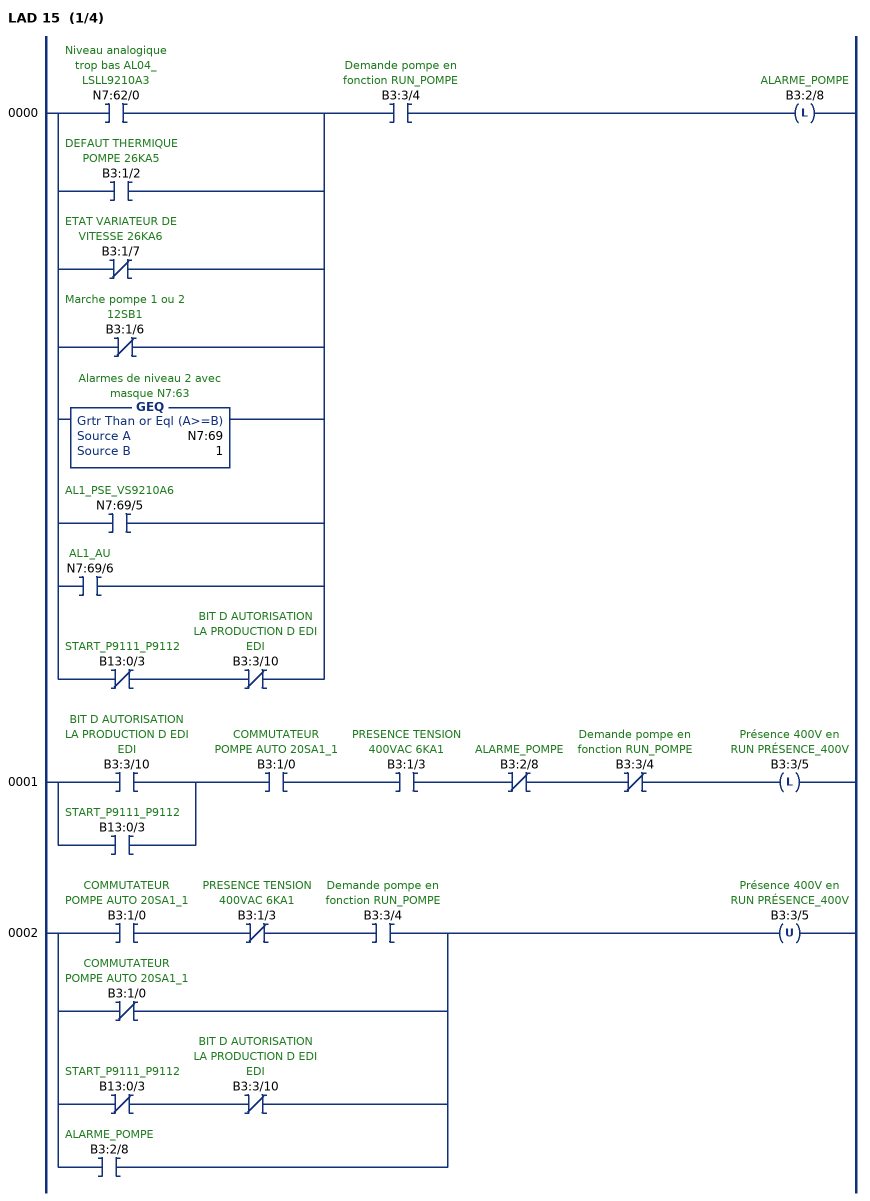
% Rung: 0 %
SOR BST XIC N7:62/0 NXB XIC B3:1/2 NXB XIO B3:1/7 NXB XIO B3:1/6 NXB GEQ N7:69 1 NXB XIC N7:69/5 NXB XIC N7:69/6 NXB XIO B13:0/3 XIO B3:3/10 BND XIC B3:3/4 OTL B3:2/8 EOR
%   N7:62/0  AL04_LSLL9210A3  "Niveau analogique trop bas" %
%   B3:1/2  26KA5  "DEFAUT THERMIQUE POMPE" %
%   B3:1/7  26KA6  "ETAT VARIATEUR DE VITESSE" %
%   B3:1/6  12SB1  "Marche pompe 1 ou 2" %
%   N7:69  "Alarmes de niveau 2 avec masque N7:63" %
%   N7:69/5  AL1_PSE_VS9210A6 %
%   N7:69/6  AL1_AU %
%   B13:0/3  START_P9111_P9112 %
%   B3:3/10  EDI  "BIT D AUTORISATION LA PRODUCTION D EDI" %
%   B3:3/4  RUN_POMPE  "Demande pompe en fonction" %
%   B3:2/8  ALARME_POMPE %
% Rung: 1 %
SOR BST XIC B3:3/10 NXB XIC B13:0/3 BND XIC B3:1/0 XIC B3:1/3 XIO B3:2/8 XIO B3:3/4 OTL B3:3/5 EOR
%   B3:3/10  EDI  "BIT D AUTORISATION LA PRODUCTION D EDI" %
%   B13:0/3  START_P9111_P9112 %
%   B3:1/0  20SA1_1  "COMMUTATEUR POMPE AUTO" %
%   B3:1/3  6KA1  "PRESENCE TENSION 400VAC" %
%   B3:2/8  ALARME_POMPE %
%   B3:3/4  RUN_POMPE  "Demande pompe en fonction" %
%   B3:3/5  PRÉSENCE_400V  "Présence 400V en RUN" %
% Rung: 2 %
SOR BST XIC B3:1/0 XIO B3:1/3 XIC B3:3/4 NXB XIO B3:1/0 NXB XIO B13:0/3 XIO B3:3/10 NXB XIC B3:2/8 BND OTU B3:3/5 EOR
%   B3:1/0  20SA1_1  "COMMUTATEUR POMPE AUTO" %
%   B3:1/3  6KA1  "PRESENCE TENSION 400VAC" %
%   B3:3/4  RUN_POMPE  "Demande pompe en fonction" %
%   B13:0/3  START_P9111_P9112 %
%   B3:3/10  EDI  "BIT D AUTORISATION LA PRODUCTION D EDI" %
%   B3:2/8  ALARME_POMPE %
%   B3:3/5  PRÉSENCE_400V  "Présence 400V en RUN" %

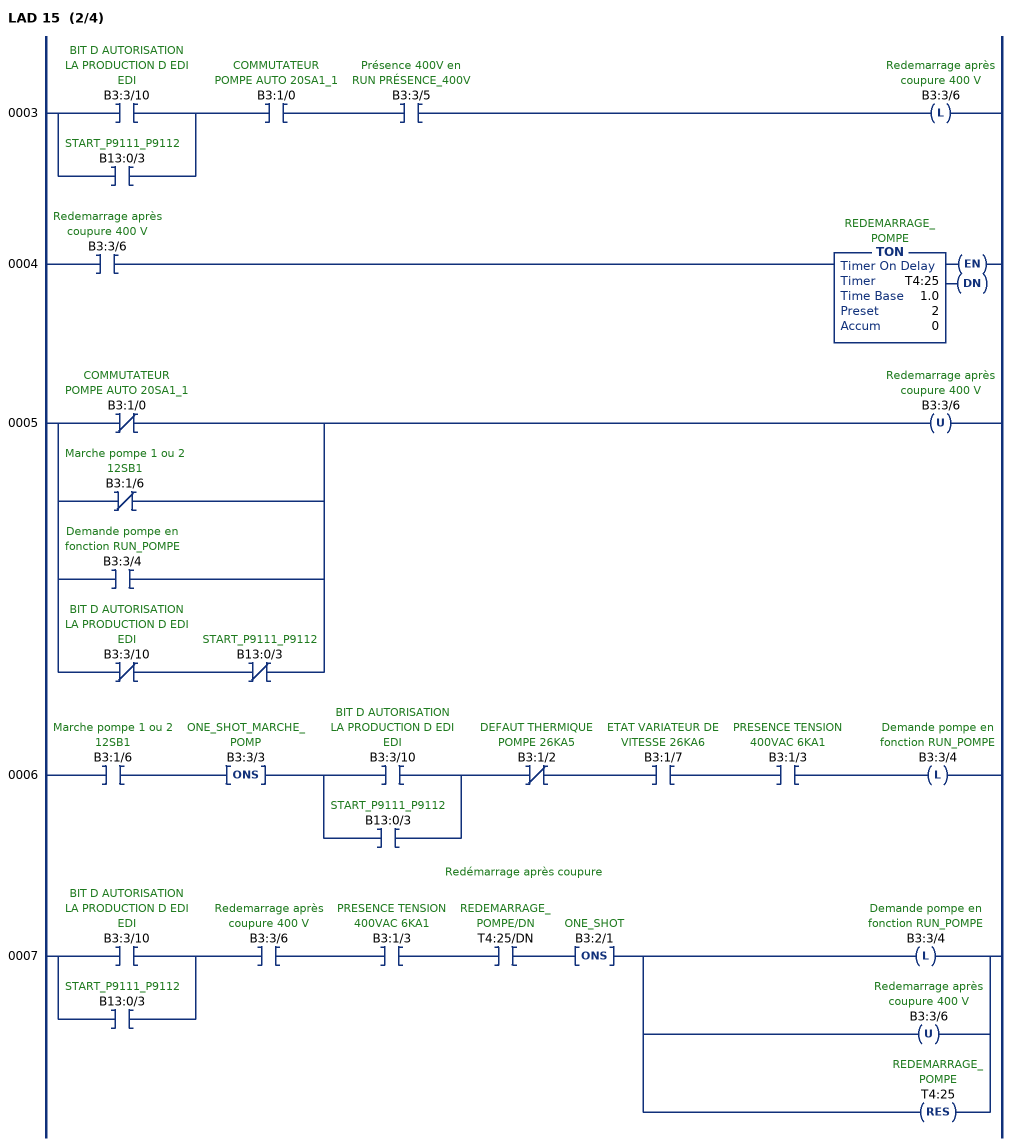
% Rung: 3 %
SOR BST XIC B3:3/10 NXB XIC B13:0/3 BND XIC B3:1/0 XIC B3:3/5 OTL B3:3/6 EOR
%   B3:3/10  EDI  "BIT D AUTORISATION LA PRODUCTION D EDI" %
%   B13:0/3  START_P9111_P9112 %
%   B3:1/0  20SA1_1  "COMMUTATEUR POMPE AUTO" %
%   B3:3/5  PRÉSENCE_400V  "Présence 400V en RUN" %
%   B3:3/6  "Redemarrage après coupure 400 V" %
% Rung: 4 %
SOR XIC B3:3/6 TON T4:25 1.0 2 0 EOR
%   B3:3/6  "Redemarrage après coupure 400 V" %
%   T4:25  REDEMARRAGE_POMPE %
% Rung: 5 %
SOR BST XIO B3:1/0 NXB XIO B3:1/6 NXB XIC B3:3/4 NXB XIO B3:3/10 XIO B13:0/3 BND OTU B3:3/6 EOR
%   B3:1/0  20SA1_1  "COMMUTATEUR POMPE AUTO" %
%   B3:1/6  12SB1  "Marche pompe 1 ou 2" %
%   B3:3/4  RUN_POMPE  "Demande pompe en fonction" %
%   B3:3/10  EDI  "BIT D AUTORISATION LA PRODUCTION D EDI" %
%   B13:0/3  START_P9111_P9112 %
%   B3:3/6  "Redemarrage après coupure 400 V" %
% Rung: 6 %
SOR XIC B3:1/6 OSR B3:3/3 BST XIC B3:3/10 NXB XIC B13:0/3 BND XIO B3:1/2 XIC B3:1/7 XIC B3:1/3 OTL B3:3/4 EOR
%   B3:1/6  12SB1  "Marche pompe 1 ou 2" %
%   B3:3/3  ONE_SHOT_MARCHE_POMP %
%   B3:3/10  EDI  "BIT D AUTORISATION LA PRODUCTION D EDI" %
%   B13:0/3  START_P9111_P9112 %
%   B3:1/2  26KA5  "DEFAUT THERMIQUE POMPE" %
%   B3:1/7  26KA6  "ETAT VARIATEUR DE VITESSE" %
%   B3:1/3  6KA1  "PRESENCE TENSION 400VAC" %
%   B3:3/4  RUN_POMPE  "Demande pompe en fonction" %
% Rung: 7 %
% Redémarrage après coupure %
SOR BST XIC B3:3/10 NXB XIC B13:0/3 BND XIC B3:3/6 XIC B3:1/3 XIC T4:25/DN OSR B3:2/1 BST OTL B3:3/4 NXB OTU B3:3/6 NXB RES T4:25 BND EOR
%   B3:3/10  EDI  "BIT D AUTORISATION LA PRODUCTION D EDI" %
%   B13:0/3  START_P9111_P9112 %
%   B3:3/6  "Redemarrage après coupure 400 V" %
%   B3:1/3  6KA1  "PRESENCE TENSION 400VAC" %
%   T4:25  REDEMARRAGE_POMPE %
%   B3:2/1  ONE_SHOT %
%   B3:3/4  RUN_POMPE  "Demande pompe en fonction" %

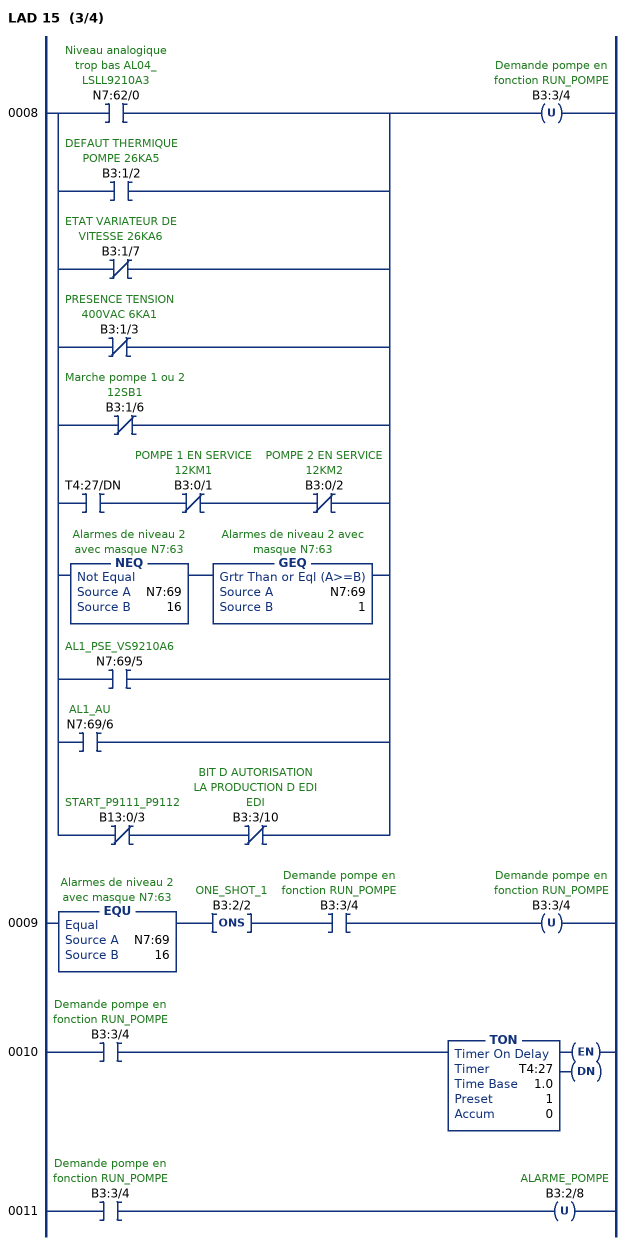
% Rung: 8 %
SOR BST XIC N7:62/0 NXB XIC B3:1/2 NXB XIO B3:1/7 NXB XIO B3:1/3 NXB XIO B3:1/6 NXB XIC T4:27/DN XIO B3:0/1 XIO B3:0/2 NXB NEQ N7:69 16 GEQ N7:69 1 NXB XIC N7:69/5 NXB XIC N7:69/6 NXB XIO B13:0/3 XIO B3:3/10 BND OTU B3:3/4 EOR
%   N7:62/0  AL04_LSLL9210A3  "Niveau analogique trop bas" %
%   B3:1/2  26KA5  "DEFAUT THERMIQUE POMPE" %
%   B3:1/7  26KA6  "ETAT VARIATEUR DE VITESSE" %
%   B3:1/3  6KA1  "PRESENCE TENSION 400VAC" %
%   B3:1/6  12SB1  "Marche pompe 1 ou 2" %
%   B3:0/1  12KM1  "POMPE 1 EN SERVICE" %
%   B3:0/2  12KM2  "POMPE 2 EN SERVICE" %
%   N7:69  "Alarmes de niveau 2 avec masque N7:63" %
%   N7:69/5  AL1_PSE_VS9210A6 %
%   N7:69/6  AL1_AU %
%   B13:0/3  START_P9111_P9112 %
%   B3:3/10  EDI  "BIT D AUTORISATION LA PRODUCTION D EDI" %
%   B3:3/4  RUN_POMPE  "Demande pompe en fonction" %
% Rung: 9 %
SOR EQU N7:69 16 OSR B3:2/2 XIC B3:3/4 OTU B3:3/4 EOR
%   N7:69  "Alarmes de niveau 2 avec masque N7:63" %
%   B3:2/2  ONE_SHOT_1 %
%   B3:3/4  RUN_POMPE  "Demande pompe en fonction" %
% Rung: 10 %
SOR XIC B3:3/4 TON T4:27 1.0 1 0 EOR
%   B3:3/4  RUN_POMPE  "Demande pompe en fonction" %
% Rung: 11 %
SOR XIC B3:3/4 OTU B3:2/8 EOR
%   B3:3/4  RUN_POMPE  "Demande pompe en fonction" %
%   B3:2/8  ALARME_POMPE %

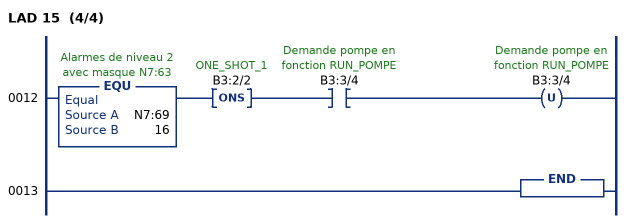
% Rung: 12 %
SOR EQU N7:69 16 OSR B3:2/2 XIC B3:3/4 OTU B3:3/4 EOR
%   N7:69  "Alarmes de niveau 2 avec masque N7:63" %
%   B3:2/2  ONE_SHOT_1 %
%   B3:3/4  RUN_POMPE  "Demande pompe en fonction" %
% Rung: 13 %
SOR END EOR

LADDER 16
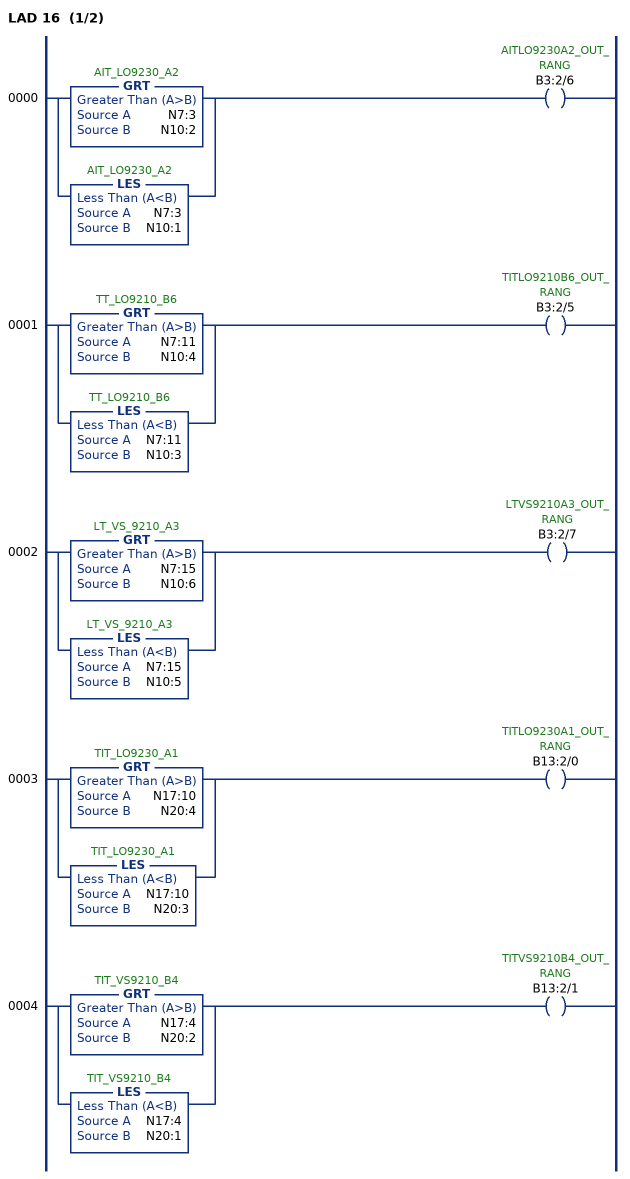
% Rung: 0 %
SOR BST GRT N7:3 N10:2 NXB LES N7:3 N10:1 BND OTE B3:2/6 EOR
%   N7:3  AIT_LO9230_A2 %
%   N10:2  OUT_RANG_MAX_AIT %
%   N10:1  OUT_RANG_MIN_AIT %
%   B3:2/6  AITLO9230A2_OUT_RANG %
% Rung: 1 %
SOR BST GRT N7:11 N10:4 NXB LES N7:11 N10:3 BND OTE B3:2/5 EOR
%   N7:11  TT_LO9210_B6 %
%   N10:4  OUT_RANG_MAX_TIT %
%   N10:3  OUT_RANG_MIN_TIT %
%   B3:2/5  TITLO9210B6_OUT_RANG %
% Rung: 2 %
SOR BST GRT N7:15 N10:6 NXB LES N7:15 N10:5 BND OTE B3:2/7 EOR
%   N7:15  LT_VS_9210_A3 %
%   N10:6  OUT_RANG_MAX_LT %
%   N10:5  OUT_RANG_MIN_LT %
%   B3:2/7  LTVS9210A3_OUT_RANG %
% Rung: 3 %
SOR BST GRT N17:10 N20:4 NXB LES N17:10 N20:3 BND OTE B13:2/0 EOR
%   N17:10  TIT_LO9230_A1 %
%   B13:2/0  TITLO9230A1_OUT_RANG %
% Rung: 4 %
SOR BST GRT N17:4 N20:2 NXB LES N17:4 N20:1 BND OTE B13:2/1 EOR
%   N17:4  TIT_VS9210_B4 %
%   B13:2/1  TITVS9210B4_OUT_RANG %

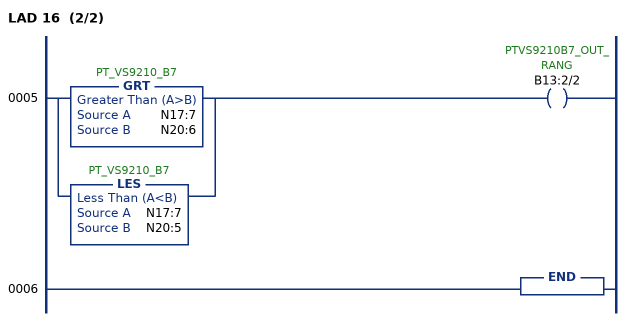
% Rung: 5 %
SOR BST GRT N17:7 N20:6 NXB LES N17:7 N20:5 BND OTE B13:2/2 EOR
%   N17:7  PT_VS9210_B7 %
%   B13:2/2  PTVS9210B7_OUT_RANG %
% Rung: 6 %
SOR END EOR

LADDER 17
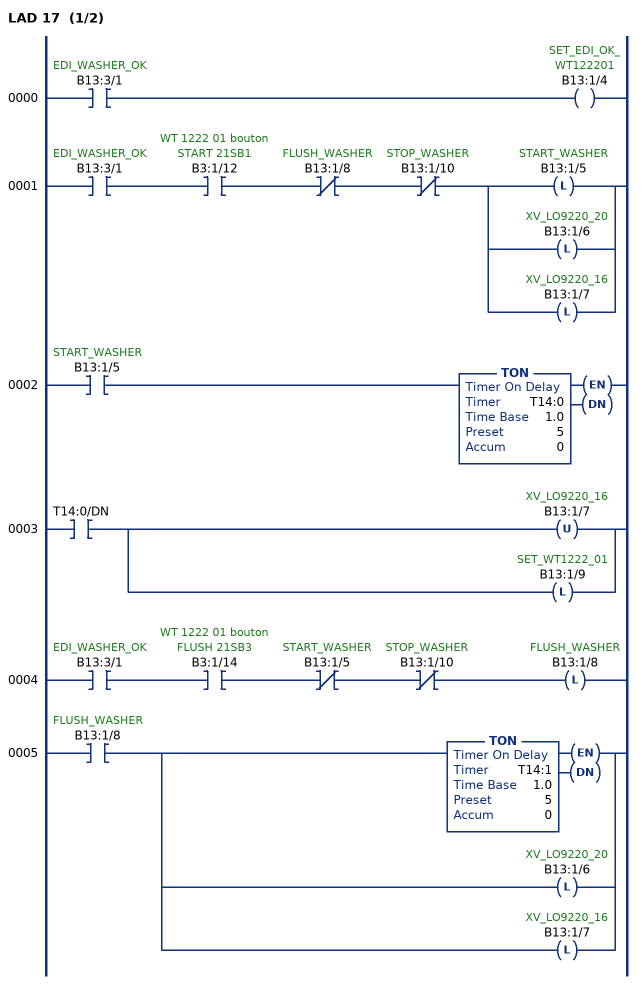
% Rung: 0 %
SOR XIC B13:3/1 OTE B13:1/4 EOR
%   B13:3/1  EDI_WASHER_OK %
%   B13:1/4  SET_EDI_OK_WT122201 %
% Rung: 1 %
SOR XIC B13:3/1 XIC B3:1/12 XIO B13:1/8 XIO B13:1/10 BST OTL B13:1/5 NXB OTL B13:1/6 NXB OTL B13:1/7 BND EOR
%   B13:3/1  EDI_WASHER_OK %
%   B3:1/12  21SB1  "WT 1222 01 bouton START" %
%   B13:1/8  FLUSH_WASHER %
%   B13:1/10  STOP_WASHER %
%   B13:1/5  START_WASHER %
%   B13:1/6  XV_LO9220_20 %
%   B13:1/7  XV_LO9220_16 %
% Rung: 2 %
SOR XIC B13:1/5 TON T14:0 1.0 5 0 EOR
%   B13:1/5  START_WASHER %
% Rung: 3 %
SOR XIC T14:0/DN BST OTU B13:1/7 NXB OTL B13:1/9 BND EOR
%   B13:1/7  XV_LO9220_16 %
%   B13:1/9  SET_WT1222_01 %
% Rung: 4 %
SOR XIC B13:3/1 XIC B3:1/14 XIO B13:1/5 XIO B13:1/10 OTL B13:1/8 EOR
%   B13:3/1  EDI_WASHER_OK %
%   B3:1/14  21SB3  "WT 1222 01 bouton FLUSH" %
%   B13:1/5  START_WASHER %
%   B13:1/10  STOP_WASHER %
%   B13:1/8  FLUSH_WASHER %
% Rung: 5 %
SOR XIC B13:1/8 BST TON T14:1 1.0 5 0 NXB OTL B13:1/6 NXB OTL B13:1/7 BND EOR
%   B13:1/8  FLUSH_WASHER %
%   B13:1/6  XV_LO9220_20 %
%   B13:1/7  XV_LO9220_16 %

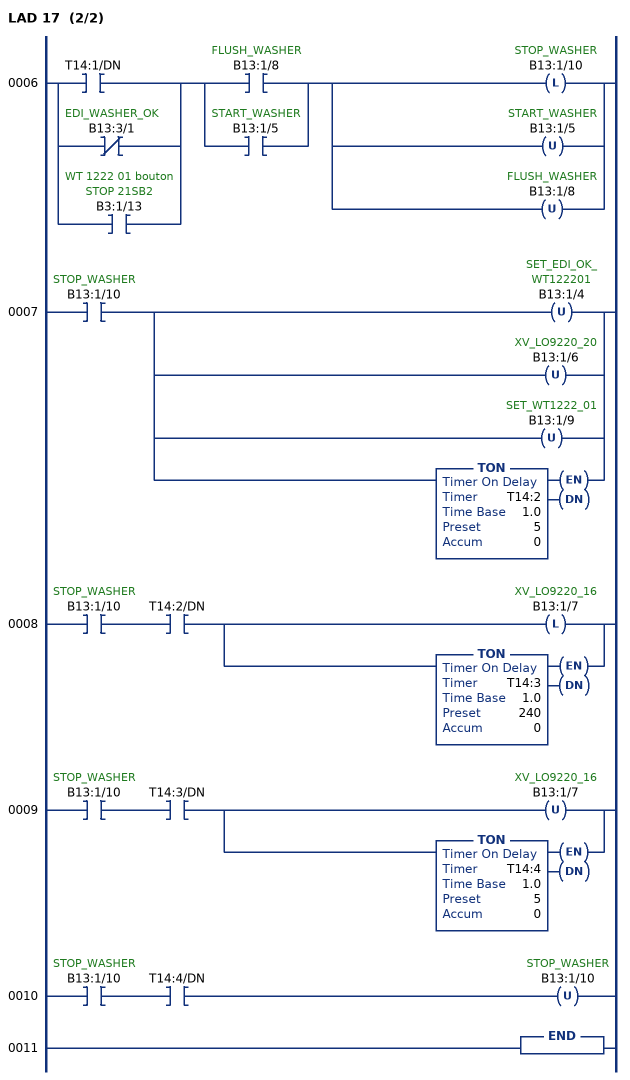
% Rung: 6 %
SOR BST XIC T14:1/DN NXB XIO B13:3/1 NXB XIC B3:1/13 BND BST XIC B13:1/8 NXB XIC B13:1/5 BND BST OTL B13:1/10 NXB OTU B13:1/5 NXB OTU B13:1/8 BND EOR
%   B13:3/1  EDI_WASHER_OK %
%   B3:1/13  21SB2  "WT 1222 01 bouton STOP" %
%   B13:1/8  FLUSH_WASHER %
%   B13:1/5  START_WASHER %
%   B13:1/10  STOP_WASHER %
% Rung: 7 %
SOR XIC B13:1/10 BST OTU B13:1/4 NXB OTU B13:1/6 NXB OTU B13:1/9 NXB TON T14:2 1.0 5 0 BND EOR
%   B13:1/10  STOP_WASHER %
%   B13:1/4  SET_EDI_OK_WT122201 %
%   B13:1/6  XV_LO9220_20 %
%   B13:1/9  SET_WT1222_01 %
% Rung: 8 %
SOR XIC B13:1/10 XIC T14:2/DN BST OTL B13:1/7 NXB TON T14:3 1.0 240 0 BND EOR
%   B13:1/10  STOP_WASHER %
%   B13:1/7  XV_LO9220_16 %
% Rung: 9 %
SOR XIC B13:1/10 XIC T14:3/DN BST OTU B13:1/7 NXB TON T14:4 1.0 5 0 BND EOR
%   B13:1/10  STOP_WASHER %
%   B13:1/7  XV_LO9220_16 %
% Rung: 10 %
SOR XIC B13:1/10 XIC T14:4/DN OTU B13:1/10 EOR
%   B13:1/10  STOP_WASHER %
% Rung: 11 %
SOR END EOR

LADDER 18
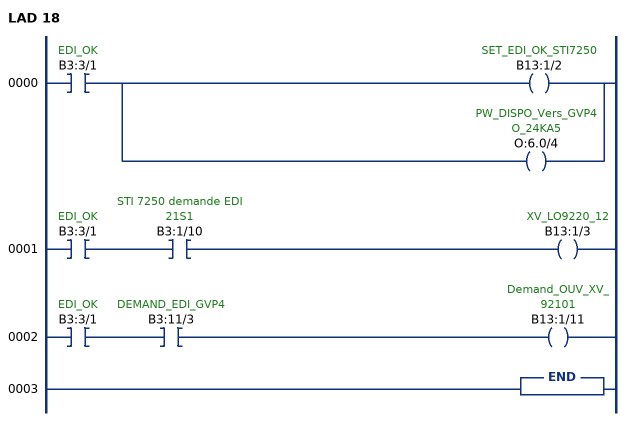
% Rung: 0 %
SOR XIC B3:3/1 BST OTE B13:1/2 NXB OTE O:6.0/4 BND EOR
%   B3:3/1  EDI_OK %
%   B13:1/2  SET_EDI_OK_STI7250 %
%   O:6.0/4  O_24KA5  "PW_DISPO_Vers_GVP4" %
% Rung: 1 %
SOR XIC B3:3/1 XIC B3:1/10 OTE B13:1/3 EOR
%   B3:3/1  EDI_OK %
%   B3:1/10  21S1  "STI 7250 demande EDI" %
%   B13:1/3  XV_LO9220_12 %
% Rung: 2 %
SOR XIC B3:3/1 XIC B3:11/3 OTE B13:1/11 EOR
%   B3:3/1  EDI_OK %
%   B3:11/3  "DEMAND_EDI_GVP4" %
%   B13:1/11  "Demand_OUV_XV_92101" %
% Rung: 3 %
SOR END EOR

LADDER 19
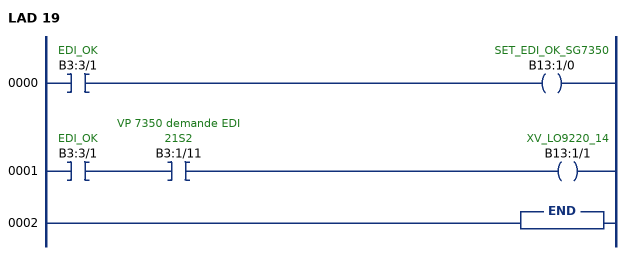
% Rung: 0 %
SOR XIC B3:3/1 OTE B13:1/0 EOR
%   B3:3/1  EDI_OK %
%   B13:1/0  SET_EDI_OK_SG7350 %
% Rung: 1 %
SOR XIC B3:3/1 XIC B3:1/11 OTE B13:1/1 EOR
%   B3:3/1  EDI_OK %
%   B3:1/11  21S2  "VP 7350 demande EDI" %
%   B13:1/1  XV_LO9220_14 %
% Rung: 2 %
SOR END EOR

LADDER 21
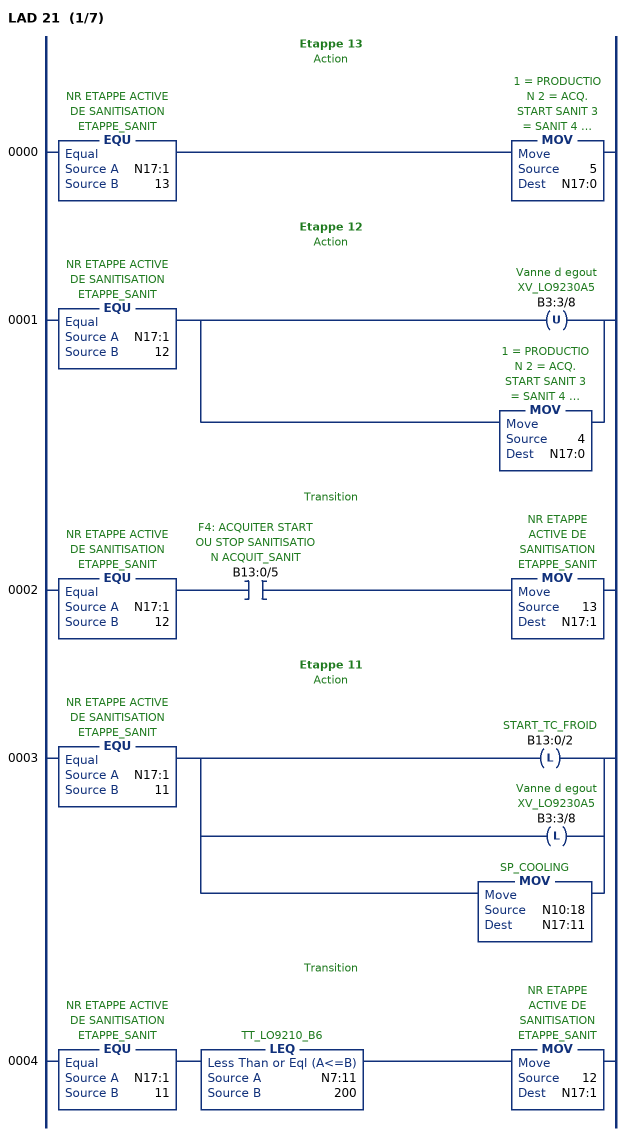
% Rung: 0 %
% TITLE: Etappe 13 %
% Action %
SOR EQU N17:1 13 MOV 5 N17:0 EOR
%   N17:1  ETAPPE_SANIT  "NR ETAPPE ACTIVE DE SANITISATION" %
%   N17:0  MODE  "1 = PRODUCTION 2 = ACQ. START SANIT 3 = SANIT 4 = ACQ. STOP SANIT 5 = FIN DE SANIT" %
% Rung: 1 %
% TITLE: Etappe 12 %
% Action %
SOR EQU N17:1 12 BST OTU B3:3/8 NXB MOV 4 N17:0 BND EOR
%   N17:1  ETAPPE_SANIT  "NR ETAPPE ACTIVE DE SANITISATION" %
%   B3:3/8  XV_LO9230A5  "Vanne d egout" %
%   N17:0  MODE  "1 = PRODUCTION 2 = ACQ. START SANIT 3 = SANIT 4 = ACQ. STOP SANIT 5 = FIN DE SANIT" %
% Rung: 2 %
% Transition %
SOR EQU N17:1 12 XIC B13:0/5 MOV 13 N17:1 EOR
%   N17:1  ETAPPE_SANIT  "NR ETAPPE ACTIVE DE SANITISATION" %
%   B13:0/5  ACQUIT_SANIT  "F4: ACQUITER START OU STOP SANITISATION" %
% Rung: 3 %
% TITLE: Etappe 11 %
% Action %
SOR EQU N17:1 11 BST OTL B13:0/2 NXB OTL B3:3/8 NXB MOV N10:18 N17:11 BND EOR
%   N17:1  ETAPPE_SANIT  "NR ETAPPE ACTIVE DE SANITISATION" %
%   B13:0/2  START_TC_FROID %
%   B3:3/8  XV_LO9230A5  "Vanne d egout" %
%   N10:18  SP_TEMP_PROD %
%   N17:11  SP_COOLING %
% Rung: 4 %
% Transition %
SOR EQU N17:1 11 LEQ N7:11 200 MOV 12 N17:1 EOR
%   N17:1  ETAPPE_SANIT  "NR ETAPPE ACTIVE DE SANITISATION" %
%   N7:11  TT_LO9210_B6 %

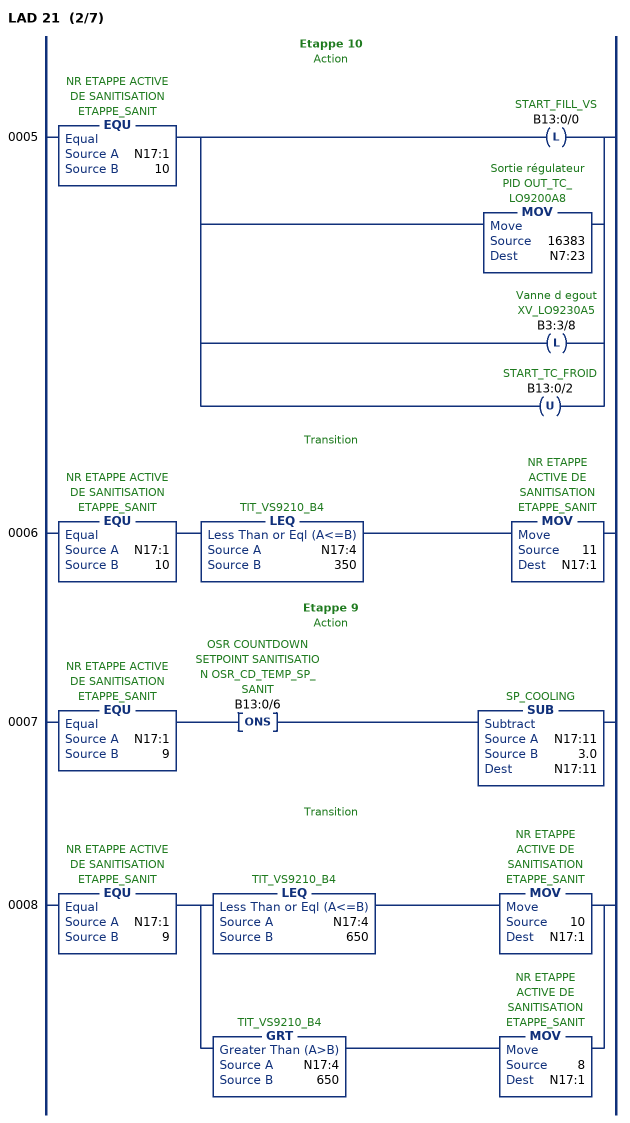
% Rung: 5 %
% TITLE: Etappe 10 %
% Action %
SOR EQU N17:1 10 BST OTL B13:0/0 NXB MOV 16383 N7:23 NXB OTL B3:3/8 NXB OTU B13:0/2 BND EOR
%   N17:1  ETAPPE_SANIT  "NR ETAPPE ACTIVE DE SANITISATION" %
%   B13:0/0  START_FILL_VS %
%   N7:23  OUT_TC_LO9200A8  "Sortie régulateur PID" %
%   B3:3/8  XV_LO9230A5  "Vanne d egout" %
%   B13:0/2  START_TC_FROID %
% Rung: 6 %
% Transition %
SOR EQU N17:1 10 LEQ N17:4 350 MOV 11 N17:1 EOR
%   N17:1  ETAPPE_SANIT  "NR ETAPPE ACTIVE DE SANITISATION" %
%   N17:4  TIT_VS9210_B4 %
% Rung: 7 %
% TITLE: Etappe 9 %
% Action %
SOR EQU N17:1 9 OSR B13:0/6 SUB N17:11 3.0 N17:11 EOR
%   N17:1  ETAPPE_SANIT  "NR ETAPPE ACTIVE DE SANITISATION" %
%   B13:0/6  OSR_CD_TEMP_SP_SANIT  "OSR COUNTDOWN SETPOINT SANITISATION" %
%   N17:11  SP_COOLING %
% Rung: 8 %
% Transition %
SOR EQU N17:1 9 BST LEQ N17:4 650 MOV 10 N17:1 NXB GRT N17:4 650 MOV 8 N17:1 BND EOR
%   N17:1  ETAPPE_SANIT  "NR ETAPPE ACTIVE DE SANITISATION" %
%   N17:4  TIT_VS9210_B4 %

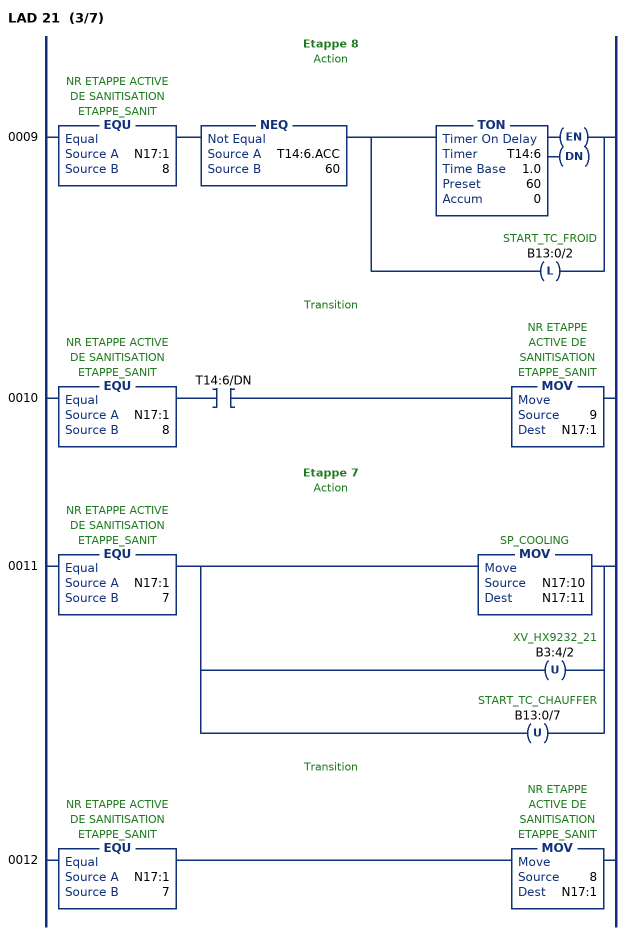
% Rung: 9 %
% TITLE: Etappe 8 %
% Action %
SOR EQU N17:1 8 NEQ T14:6.ACC 60 BST TON T14:6 1.0 60 0 NXB OTL B13:0/2 BND EOR
%   N17:1  ETAPPE_SANIT  "NR ETAPPE ACTIVE DE SANITISATION" %
%   B13:0/2  START_TC_FROID %
% Rung: 10 %
% Transition %
SOR EQU N17:1 8 XIC T14:6/DN MOV 9 N17:1 EOR
%   N17:1  ETAPPE_SANIT  "NR ETAPPE ACTIVE DE SANITISATION" %
% Rung: 11 %
% TITLE: Etappe 7 %
% Action %
SOR EQU N17:1 7 BST MOV N17:10 N17:11 NXB OTU B3:4/2 NXB OTU B13:0/7 BND EOR
%   N17:1  ETAPPE_SANIT  "NR ETAPPE ACTIVE DE SANITISATION" %
%   N17:10  TIT_LO9230_A1 %
%   N17:11  SP_COOLING %
%   B3:4/2  XV_HX9232_21 %
%   B13:0/7  START_TC_CHAUFFER %
% Rung: 12 %
% Transition %
SOR EQU N17:1 7 MOV 8 N17:1 EOR
%   N17:1  ETAPPE_SANIT  "NR ETAPPE ACTIVE DE SANITISATION" %

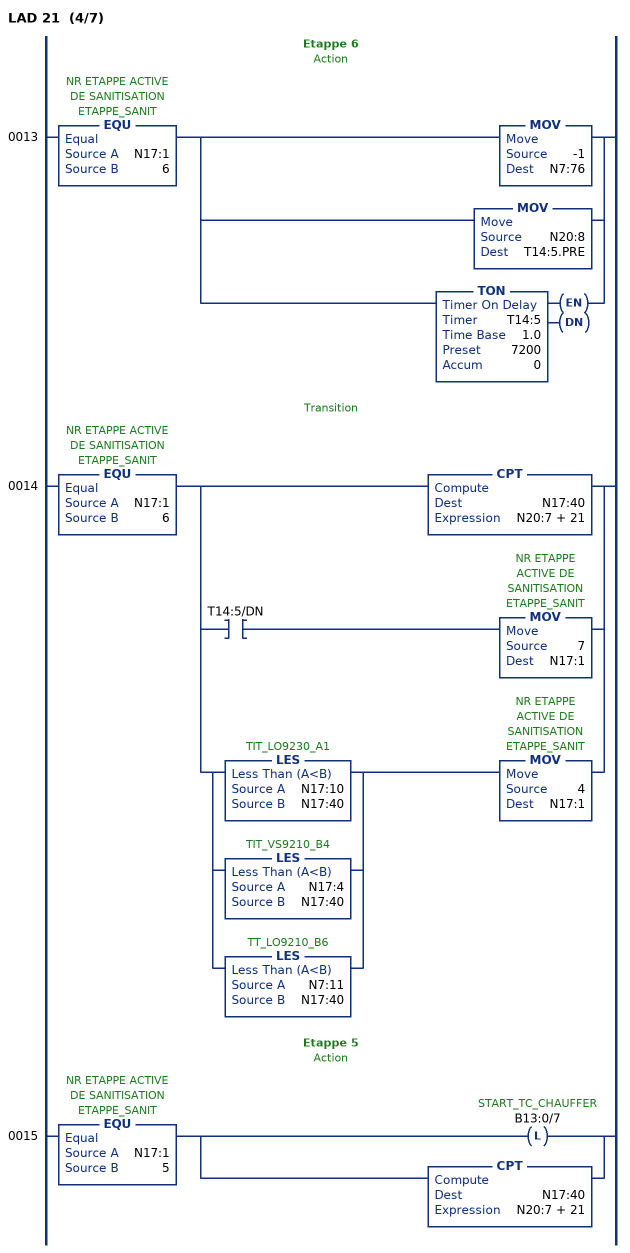
% Rung: 13 %
% TITLE: Etappe 6 %
% Action %
SOR EQU N17:1 6 BST MOV -1 N7:76 NXB MOV N20:8 T14:5.PRE NXB TON T14:5 1.0 7200 0 BND EOR
%   N17:1  ETAPPE_SANIT  "NR ETAPPE ACTIVE DE SANITISATION" %
%   N20:8  TEMPS_SANIT %
% Rung: 14 %
% Transition %
SOR EQU N17:1 6 BST CPT N17:40 " N20:7 + 21 " NXB XIC T14:5/DN MOV 7 N17:1 NXB BST LES N17:10 N17:40 NXB LES N17:4 N17:40 NXB LES N7:11 N17:40 BND MOV 4 N17:1 BND EOR
%   N17:1  ETAPPE_SANIT  "NR ETAPPE ACTIVE DE SANITISATION" %
%   N20:7  SP_TEMP_SANIT %
%   N17:10  TIT_LO9230_A1 %
%   N17:4  TIT_VS9210_B4 %
%   N7:11  TT_LO9210_B6 %
% Rung: 15 %
% TITLE: Etappe 5 %
% Action %
SOR EQU N17:1 5 BST OTL B13:0/7 NXB CPT N17:40 " N20:7 + 21 " BND EOR
%   N17:1  ETAPPE_SANIT  "NR ETAPPE ACTIVE DE SANITISATION" %
%   B13:0/7  START_TC_CHAUFFER %
%   N20:7  SP_TEMP_SANIT %

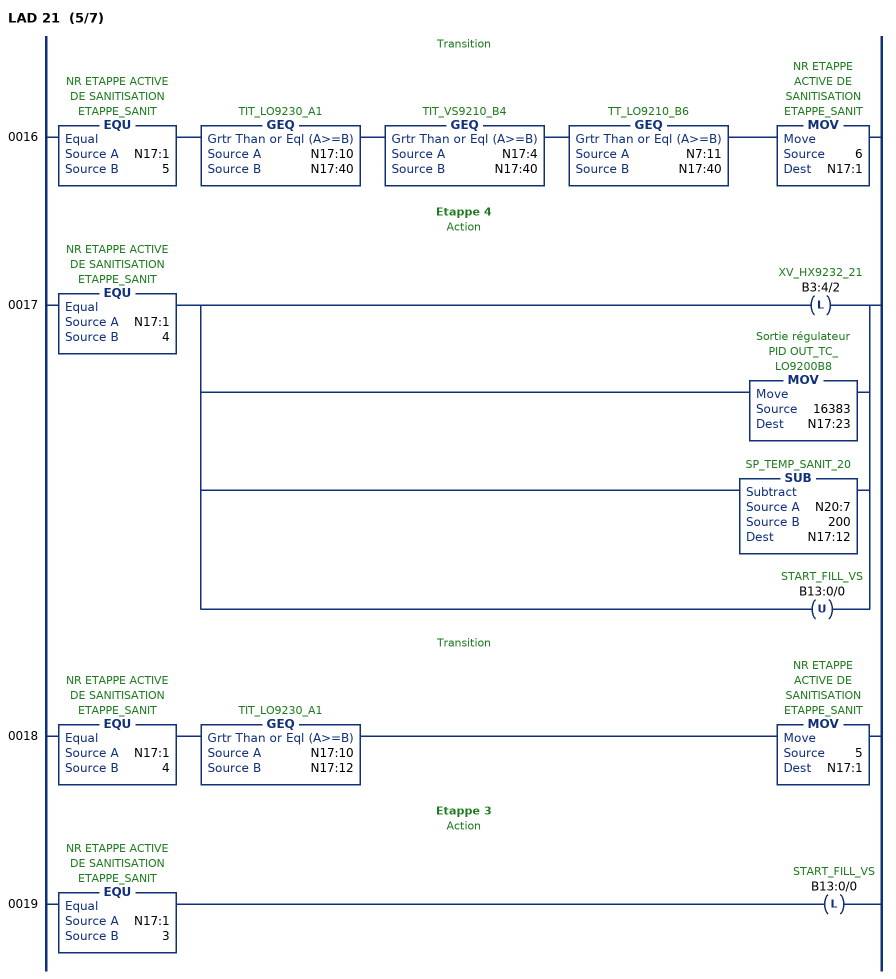
% Rung: 16 %
% Transition %
SOR EQU N17:1 5 GEQ N17:10 N17:40 GEQ N17:4 N17:40 GEQ N7:11 N17:40 MOV 6 N17:1 EOR
%   N17:1  ETAPPE_SANIT  "NR ETAPPE ACTIVE DE SANITISATION" %
%   N17:10  TIT_LO9230_A1 %
%   N17:4  TIT_VS9210_B4 %
%   N7:11  TT_LO9210_B6 %
% Rung: 17 %
% TITLE: Etappe 4 %
% Action %
SOR EQU N17:1 4 BST OTL B3:4/2 NXB MOV 16383 N17:23 NXB SUB N20:7 200 N17:12 NXB OTU B13:0/0 BND EOR
%   N17:1  ETAPPE_SANIT  "NR ETAPPE ACTIVE DE SANITISATION" %
%   B3:4/2  XV_HX9232_21 %
%   N17:23  OUT_TC_LO9200B8  "Sortie régulateur PID" %
%   N20:7  SP_TEMP_SANIT %
%   N17:12  SP_TEMP_SANIT_20 %
%   B13:0/0  START_FILL_VS %
% Rung: 18 %
% Transition %
SOR EQU N17:1 4 GEQ N17:10 N17:12 MOV 5 N17:1 EOR
%   N17:1  ETAPPE_SANIT  "NR ETAPPE ACTIVE DE SANITISATION" %
%   N17:10  TIT_LO9230_A1 %
%   N17:12  SP_TEMP_SANIT_20 %
% Rung: 19 %
% TITLE: Etappe 3 %
% Action %
SOR EQU N17:1 3 OTL B13:0/0 EOR
%   N17:1  ETAPPE_SANIT  "NR ETAPPE ACTIVE DE SANITISATION" %
%   B13:0/0  START_FILL_VS %

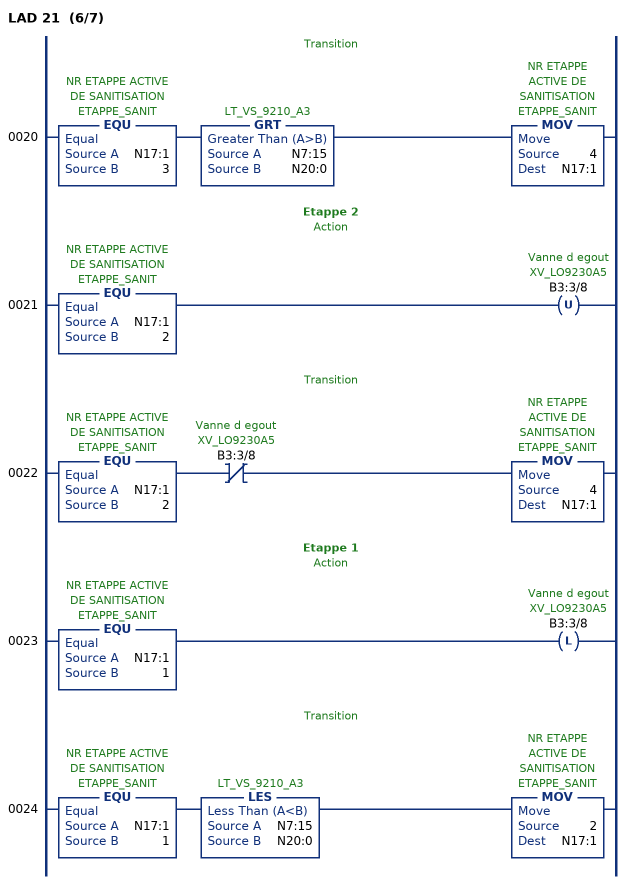
% Rung: 20 %
% Transition %
SOR EQU N17:1 3 GRT N7:15 N20:0 MOV 4 N17:1 EOR
%   N17:1  ETAPPE_SANIT  "NR ETAPPE ACTIVE DE SANITISATION" %
%   N7:15  LT_VS_9210_A3 %
%   N20:0  NIV_SANIT  "Niveau de sanitisation" %
% Rung: 21 %
% TITLE: Etappe 2 %
% Action %
SOR EQU N17:1 2 OTU B3:3/8 EOR
%   N17:1  ETAPPE_SANIT  "NR ETAPPE ACTIVE DE SANITISATION" %
%   B3:3/8  XV_LO9230A5  "Vanne d egout" %
% Rung: 22 %
% Transition %
SOR EQU N17:1 2 XIO B3:3/8 MOV 4 N17:1 EOR
%   N17:1  ETAPPE_SANIT  "NR ETAPPE ACTIVE DE SANITISATION" %
%   B3:3/8  XV_LO9230A5  "Vanne d egout" %
% Rung: 23 %
% TITLE: Etappe 1 %
% Action %
SOR EQU N17:1 1 OTL B3:3/8 EOR
%   N17:1  ETAPPE_SANIT  "NR ETAPPE ACTIVE DE SANITISATION" %
%   B3:3/8  XV_LO9230A5  "Vanne d egout" %
% Rung: 24 %
% Transition %
SOR EQU N17:1 1 LES N7:15 N20:0 MOV 2 N17:1 EOR
%   N17:1  ETAPPE_SANIT  "NR ETAPPE ACTIVE DE SANITISATION" %
%   N7:15  LT_VS_9210_A3 %
%   N20:0  NIV_SANIT  "Niveau de sanitisation" %

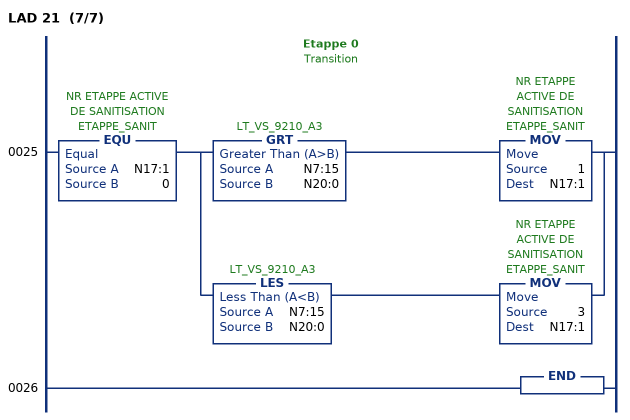
% Rung: 25 %
% TITLE: Etappe 0 %
% Transition %
SOR EQU N17:1 0 BST GRT N7:15 N20:0 MOV 1 N17:1 NXB LES N7:15 N20:0 MOV 3 N17:1 BND EOR
%   N17:1  ETAPPE_SANIT  "NR ETAPPE ACTIVE DE SANITISATION" %
%   N7:15  LT_VS_9210_A3 %
%   N20:0  NIV_SANIT  "Niveau de sanitisation" %
% Rung: 26 %
SOR END EOR

LADDER 22
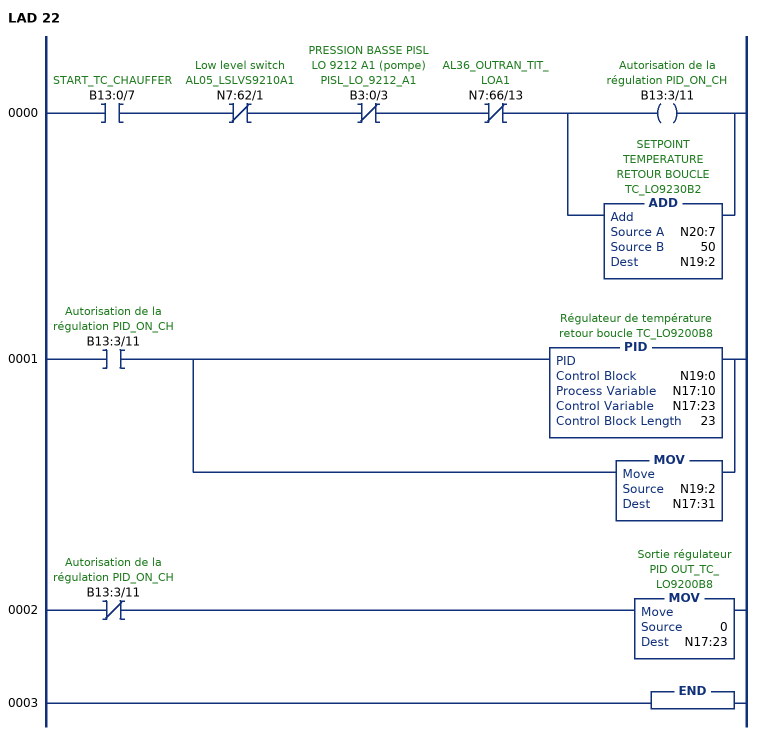
% Rung: 0 %
SOR XIC B13:0/7 XIO N7:62/1 XIO B3:0/3 XIO N7:66/13 BST OTE B13:3/11 NXB ADD N20:7 50 N19:2 BND EOR
%   B13:0/7  START_TC_CHAUFFER %
%   N7:62/1  AL05_LSLVS9210A1  "Low level switch" %
%   B3:0/3  PISL_LO_9212_A1  "PRESSION BASSE PISL LO 9212 A1 (pompe)" %
%   N7:66/13  AL36_OUTRAN_TIT_LOA1 %
%   B13:3/11  PID_ON_CH  "Autorisation de la régulation" %
%   N20:7  SP_TEMP_SANIT %
%   N19:2  TC_LO9230B2  "SETPOINT TEMPERATURE RETOUR BOUCLE" %
% Rung: 1 %
SOR XIC B13:3/11 BST PID N19:0 N17:10 N17:23 23 NXB MOV N19:2 N17:31 BND EOR
%   B13:3/11  PID_ON_CH  "Autorisation de la régulation" %
%   N19:0  TC_LO9200B8  "Régulateur de température retour boucle" %
%   N17:10  TIT_LO9230_A1 %
%   N17:23  OUT_TC_LO9200B8  "Sortie régulateur PID" %
%   N19:2  TC_LO9230B2  "SETPOINT TEMPERATURE RETOUR BOUCLE" %
% Rung: 2 %
SOR XIO B13:3/11 MOV 0 N17:23 EOR
%   B13:3/11  PID_ON_CH  "Autorisation de la régulation" %
%   N17:23  OUT_TC_LO9200B8  "Sortie régulateur PID" %
% Rung: 3 %
SOR END EOR

LADDER 23
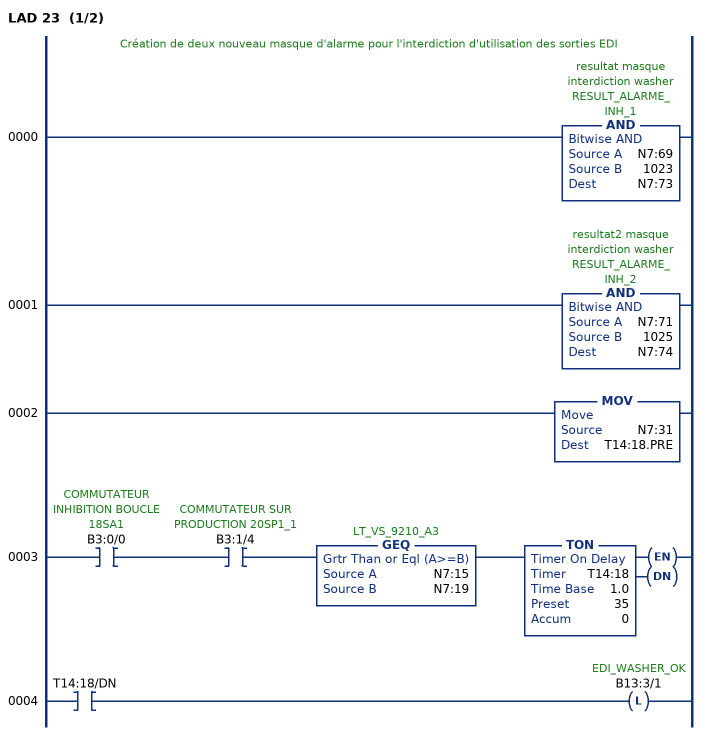
% Rung: 0 %
% Création de deux nouveau masque d'alarme pour l'interdiction d'utilisation des sorties EDI %
SOR AND N7:69 1023 N7:73 EOR
%   N7:69  "Alarmes de niveau 2 avec masque N7:63" %
%   N7:73  RESULT_ALARME_INH_1  "resultat masque interdiction washer" %
% Rung: 1 %
SOR AND N7:71 1025 N7:74 EOR
%   N7:71  "Alarmes de niveau 3/2 avec masque N7:67" %
%   N7:74  RESULT_ALARME_INH_2  "resultat2 masque interdiction washer" %
% Rung: 2 %
SOR MOV N7:31 T14:18.PRE EOR
%   N7:31  TEMPO_WASHER %
% Rung: 3 %
SOR XIC B3:0/0 XIC B3:1/4 GEQ N7:15 N7:19 TON T14:18 1.0 35 0 EOR
%   B3:0/0  18SA1  "COMMUTATEUR INHIBITION BOUCLE" %
%   B3:1/4  20SP1_1  "COMMUTATEUR SUR PRODUCTION" %
%   N7:15  LT_VS_9210_A3 %
%   N7:19  LSM_VS9210_A3_2 %
% Rung: 4 %
SOR XIC T14:18/DN OTL B13:3/1 EOR
%   B13:3/1  EDI_WASHER_OK %

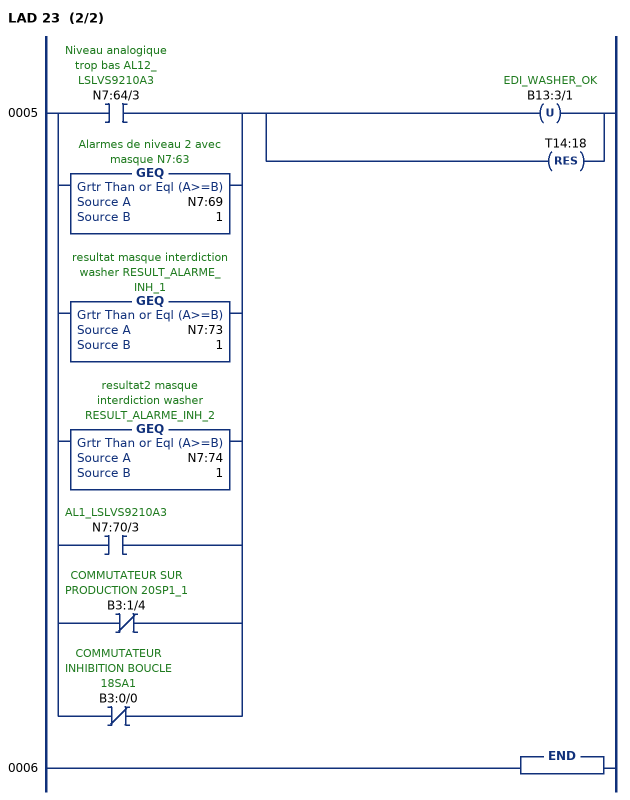
% Rung: 5 %
SOR BST XIC N7:64/3 NXB GEQ N7:69 1 NXB GEQ N7:73 1 NXB GEQ N7:74 1 NXB XIC N7:70/3 NXB XIO B3:1/4 NXB XIO B3:0/0 BND BST OTU B13:3/1 NXB RES T14:18 BND EOR
%   N7:64/3  AL12_LSLVS9210A3  "Niveau analogique trop bas" %
%   N7:69  "Alarmes de niveau 2 avec masque N7:63" %
%   N7:73  RESULT_ALARME_INH_1  "resultat masque interdiction washer" %
%   N7:74  RESULT_ALARME_INH_2  "resultat2 masque interdiction washer" %
%   N7:70/3  AL1_LSLVS9210A3 %
%   B3:1/4  20SP1_1  "COMMUTATEUR SUR PRODUCTION" %
%   B3:0/0  18SA1  "COMMUTATEUR INHIBITION BOUCLE" %
%   B13:3/1  EDI_WASHER_OK %
% Rung: 6 %
SOR END EOR

LADDER 24
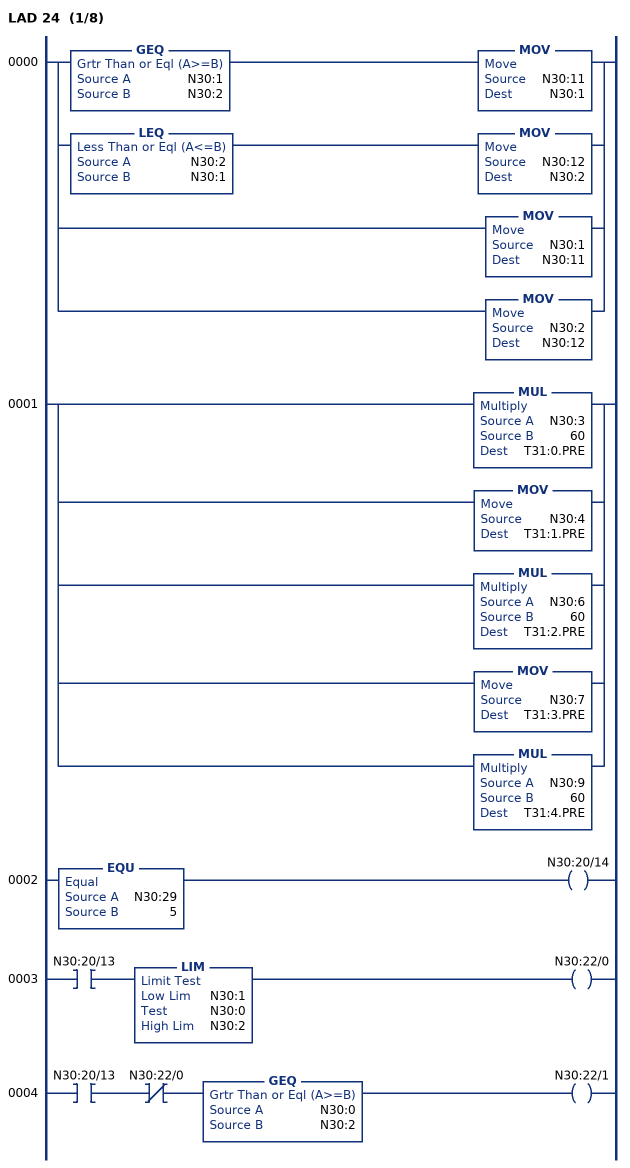
% Rung: 0 %
SOR BST GEQ N30:1 N30:2 MOV N30:11 N30:1 NXB LEQ N30:2 N30:1 MOV N30:12 N30:2 NXB MOV N30:1 N30:11 NXB MOV N30:2 N30:12 BND EOR
% Rung: 1 %
SOR BST MUL N30:3 60 T31:0.PRE NXB MOV N30:4 T31:1.PRE NXB MUL N30:6 60 T31:2.PRE NXB MOV N30:7 T31:3.PRE NXB MUL N30:9 60 T31:4.PRE BND EOR
% Rung: 2 %
SOR EQU N30:29 5 OTE N30:20/14 EOR
% Rung: 3 %
SOR XIC N30:20/13 LIM N30:1 N30:0 N30:2 OTE N30:22/0 EOR
% Rung: 4 %
SOR XIC N30:20/13 XIO N30:22/0 GEQ N30:0 N30:2 OTE N30:22/1 EOR

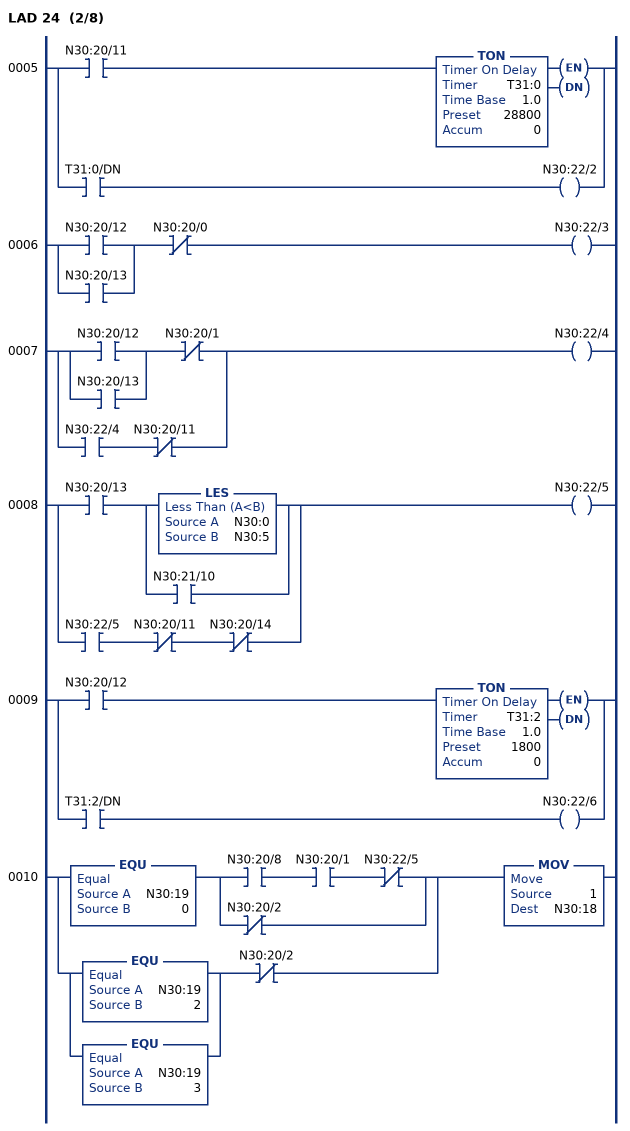
% Rung: 5 %
SOR BST XIC N30:20/11 TON T31:0 1.0 28800 0 NXB XIC T31:0/DN OTE N30:22/2 BND EOR
% Rung: 6 %
SOR BST XIC N30:20/12 NXB XIC N30:20/13 BND XIO N30:20/0 OTE N30:22/3 EOR
% Rung: 7 %
SOR BST BST XIC N30:20/12 NXB XIC N30:20/13 BND XIO N30:20/1 NXB XIC N30:22/4 XIO N30:20/11 BND OTE N30:22/4 EOR
% Rung: 8 %
SOR BST XIC N30:20/13 BST LES N30:0 N30:5 NXB XIC N30:21/10 BND NXB XIC N30:22/5 XIO N30:20/11 XIO N30:20/14 BND OTE N30:22/5 EOR
% Rung: 9 %
SOR BST XIC N30:20/12 TON T31:2 1.0 1800 0 NXB XIC T31:2/DN OTE N30:22/6 BND EOR
% Rung: 10 %
SOR BST EQU N30:19 0 BST XIC N30:20/8 XIC N30:20/1 XIO N30:22/5 NXB XIO N30:20/2 BND NXB BST EQU N30:19 2 NXB EQU N30:19 3 BND XIO N30:20/2 BND MOV 1 N30:18 EOR

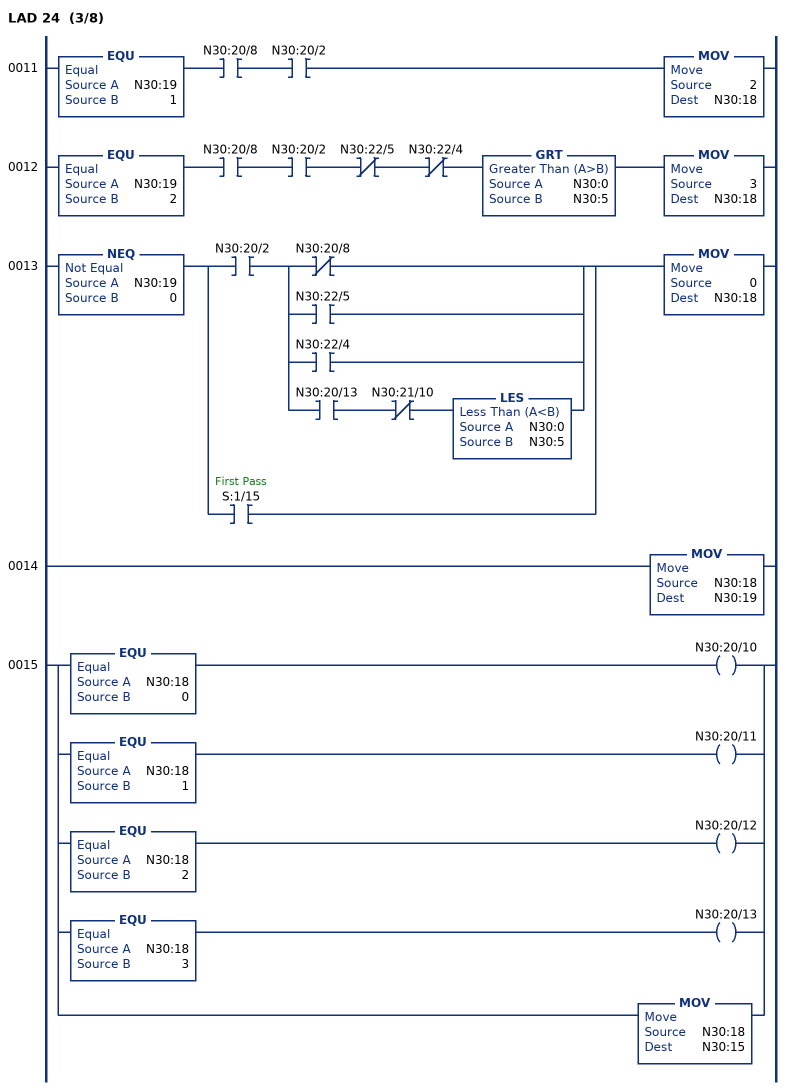
% Rung: 11 %
SOR EQU N30:19 1 XIC N30:20/8 XIC N30:20/2 MOV 2 N30:18 EOR
% Rung: 12 %
SOR EQU N30:19 2 XIC N30:20/8 XIC N30:20/2 XIO N30:22/5 XIO N30:22/4 GRT N30:0 N30:5 MOV 3 N30:18 EOR
% Rung: 13 %
SOR NEQ N30:19 0 BST XIC N30:20/2 BST XIO N30:20/8 NXB XIC N30:22/5 NXB XIC N30:22/4 NXB XIC N30:20/13 XIO N30:21/10 LES N30:0 N30:5 BND NXB XIC S:1/15 BND MOV 0 N30:18 EOR
%   S:1/15  "First Pass" %
% Rung: 14 %
SOR MOV N30:18 N30:19 EOR
% Rung: 15 %
SOR BST EQU N30:18 0 OTE N30:20/10 NXB EQU N30:18 1 OTE N30:20/11 NXB EQU N30:18 2 OTE N30:20/12 NXB EQU N30:18 3 OTE N30:20/13 NXB MOV N30:18 N30:15 BND EOR

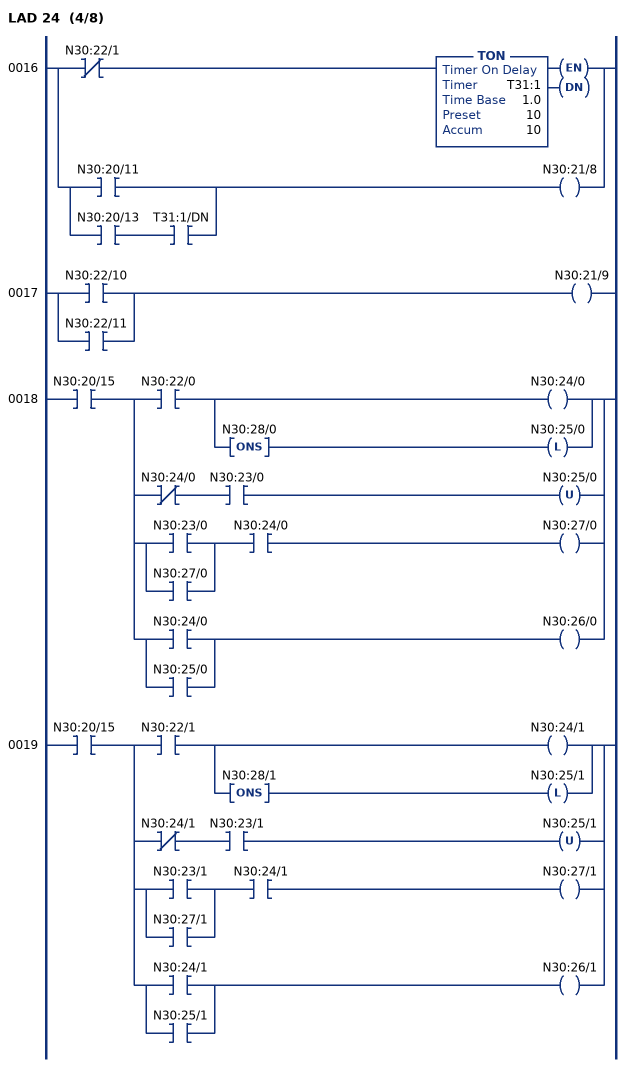
% Rung: 16 %
SOR BST XIO N30:22/1 TON T31:1 1.0 10 10 NXB BST XIC N30:20/11 NXB XIC N30:20/13 XIC T31:1/DN BND OTE N30:21/8 BND EOR
% Rung: 17 %
SOR BST XIC N30:22/10 NXB XIC N30:22/11 BND OTE N30:21/9 EOR
% Rung: 18 %
SOR XIC N30:20/15 BST XIC N30:22/0 BST OTE N30:24/0 NXB OSR N30:28/0 OTL N30:25/0 BND NXB XIO N30:24/0 XIC N30:23/0 OTU N30:25/0 NXB BST XIC N30:23/0 NXB XIC N30:27/0 BND XIC N30:24/0 OTE N30:27/0 NXB BST XIC N30:24/0 NXB XIC N30:25/0 BND OTE N30:26/0 BND EOR
% Rung: 19 %
SOR XIC N30:20/15 BST XIC N30:22/1 BST OTE N30:24/1 NXB OSR N30:28/1 OTL N30:25/1 BND NXB XIO N30:24/1 XIC N30:23/1 OTU N30:25/1 NXB BST XIC N30:23/1 NXB XIC N30:27/1 BND XIC N30:24/1 OTE N30:27/1 NXB BST XIC N30:24/1 NXB XIC N30:25/1 BND OTE N30:26/1 BND EOR

